Staubli VAL3: iState.pgx

public program iState(num& nNum[] (dimensions=1))
begin
end
